// TIA Portal V19 export
VAR_GLOBAL   // PLC tag table "DefaultTagTable"
   Tag_1 AT %M20.7 : Bool;
END_VAR
